# EPICS autosave request: dxp/branches/R3-0-branch/dxpApp/Db/dxpMED_settings.req
$(P)PresetReal
$(P)PresetLive
$(P)StatusAll.SCAN
$(P)ReadAll.SCAN
$(P)TraceTimes
$(P)TraceModes
$(P)EnableClientWait
